TYPE ST_ConfigurableCylinderOutImm :
STRUCT
    Position   : E_CylinderPosition;
    AtHome     : BOOL;
    AtWork     : BOOL;
    Diagnostic : ST_Diagnostic;
END_STRUCT
END_TYPE

(* stored: Version 1.1.0.1, ProductVersion 3.1.4024.12
   DUT ST_ConfigurableCylinderOutImm: Id {ba801215-4aaa-44e5-85e9-e148140b79a5} *)
